ABB RAPID module: CalibData.mod

MODULE CalibData
    PERS tooldata tWeldGun:=[TRUE,[[125.800591275,0,391.268161315],[0.898794046,0,0.438371147,0]],[3,[0,0,100],[0,1,0,0],0,0,0]];
    PERS tooldata pen:=[TRUE,[[0,0,139],[1,0,0,0]],[0.5,[0,0,20],[1,0,0,0],0,0,0]];
    TASK PERS wobjdata Workobject_Paper:=[FALSE,TRUE,"",[[450,125,118],[0,1,0,0]],[[50,50,0],[1,0,0,0]]];

    CONST robtarget Origem:=[[-50,-50,-2.5],[1,0,0,0],[0,0,0,0],[9E+09,9E+09,9E+09,9E+09,9E+09,9E+09]];
    CONST robtarget Default_position:=[[55,95,-102.5],[1,0,0,0],[0,0,0,0],[9E+09,9E+09,9E+09,9E+09,9E+09,9E+09]];
ENDMODULE
